// TIA Portal V21 export
VAR_GLOBAL   // PLC tag table "K_Consenso"
END_VAR
VAR_GLOBAL CONSTANT   // user constants
   K_ConsensoVerso_CFT_ImpiantoInSterilizzazione : Int := 1;
   K_ConsensoVerso_CFT_ImpiantoInLavaggio : Int := 2;
   K_ConsensoVerso_CFT_ImpulsiPompaPistoni : Int := 3;
   K_ConsensoVerso_CFT_ImpiantoInProduzione : Int := 4;
   K_ConsensoVerso_CFT_ProdottoDisponibile : Int := 5;
   K_ConsensoVerso_QCI_ChiamataProdotto : Int := 1;
   K_ConsensoDaCFT_SterilizzazioneTerminata : Int := 1;
   K_ConsensoDaCFT_SterilizzazioneInCorso : Int := 2;
   K_ConsensoDaCFT_LavaggioInCorso : Int := 3;
   K_ConsensoDaCFT_DosaggioInCorso : Int := 4;
   K_ConsensoDaCFT_RiempitriceInProduzione : Int := 5;
   K_ConsensoDaCFT_TemperaturaSterilizzazioneOk : Int := 6;
END_VAR
